(* IEC 61131-3 sources: eCockpitGit/test_project/src/%F%NormalFolder, 3 files *)

(* ---- %DUT%alias_test_1.st ---- *)
TYPE alias_test_1 : INT; END_TYPE

(* ---- %GVL%GVL_test_1.st ---- *)
{attribute 'qualified_only'}
VAR_GLOBAL
	variablssss: BOOL;
	variablssss1: INT;
	variablssss2: BOOL;
	variablssss3: STRING;
	variablssss4: union_test;
	variablssss5: BOOL;
END_VAR

(* ---- %POU%func_test_1.st ---- *)
FUNCTION func_test_1 : BOOL
VAR_INPUT
END_VAR
VAR
END_VAR

(*%!%__DELIMITER__%!%*)
